% RSLogix 500 project Multiposition-Servo-Application.RSS, saved by version 8.30.00.16 %
PROJECT "UNTITLED"    % processor: Bul.1763 MicroLogix 1100 Series B %

PROGRAM FILES
  LAD 2 "MAIN"  4 rungs
  LAD 3 "IO"  7 rungs
  LAD 4 "CTRL"  10 rungs
  LAD 5 "POSI"  9 rungs

DATA FILES
  O0 OUTPUT  4 elements
  I1 INPUT  6 elements
  S2 STATUS  66 elements
  B3 BINARY  4 elements
  T4 TIMER  3 elements
  C5 COUNTER  1 elements
  R6 CONTROL  1 elements
  N7 INTEGER  2 elements
  F8 FLOAT  1 elements

LADDER 2 "MAIN"
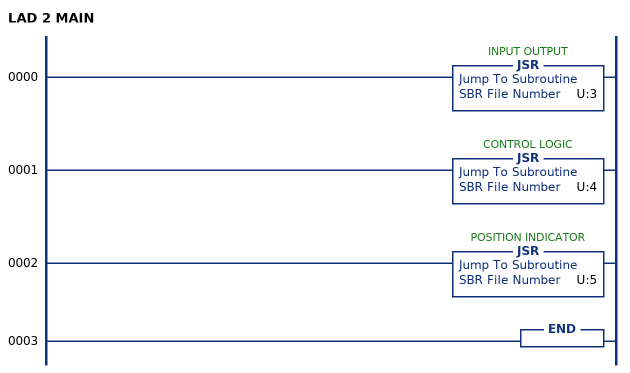
% Rung: 0 %
SOR JSR U:3 EOR
%   U:3  "INPUT OUTPUT" %
% Rung: 1 %
SOR JSR U:4 EOR
%   U:4  "CONTROL LOGIC" %
% Rung: 2 %
SOR JSR U:5 EOR
%   U:5  "POSITION INDICATOR" %
% Rung: 3 %
SOR END EOR

LADDER 3 "IO"
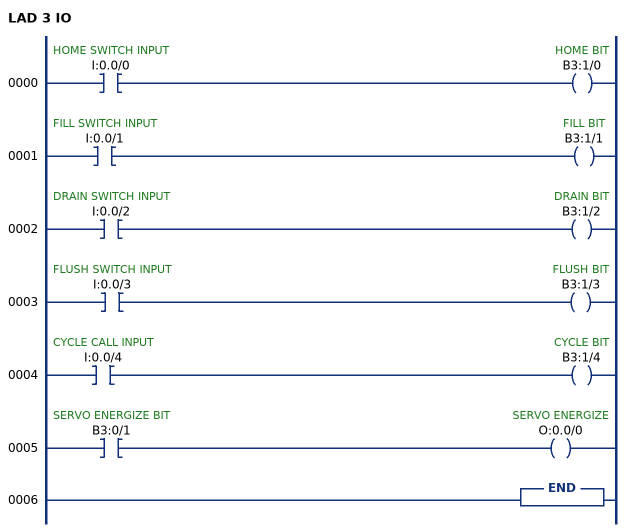
% Rung: 0 %
SOR XIC I:0.0/0 OTE B3:1/0 EOR
%   I:0.0/0  "HOME SWITCH INPUT" %
%   B3:1/0  "HOME BIT" %
% Rung: 1 %
SOR XIC I:0.0/1 OTE B3:1/1 EOR
%   I:0.0/1  "FILL SWITCH INPUT" %
%   B3:1/1  "FILL BIT" %
% Rung: 2 %
SOR XIC I:0.0/2 OTE B3:1/2 EOR
%   I:0.0/2  "DRAIN SWITCH INPUT" %
%   B3:1/2  "DRAIN BIT" %
% Rung: 3 %
SOR XIC I:0.0/3 OTE B3:1/3 EOR
%   I:0.0/3  "FLUSH SWITCH INPUT" %
%   B3:1/3  "FLUSH BIT" %
% Rung: 4 %
SOR XIC I:0.0/4 OTE B3:1/4 EOR
%   I:0.0/4  "CYCLE CALL INPUT" %
%   B3:1/4  "CYCLE BIT" %
% Rung: 5 %
SOR XIC B3:0/1 OTE O:0.0/0 EOR
%   B3:0/1  "SERVO ENERGIZE BIT" %
%   O:0.0/0  "SERVO ENERGIZE" %
% Rung: 6 %
SOR END EOR

LADDER 4 "CTRL"
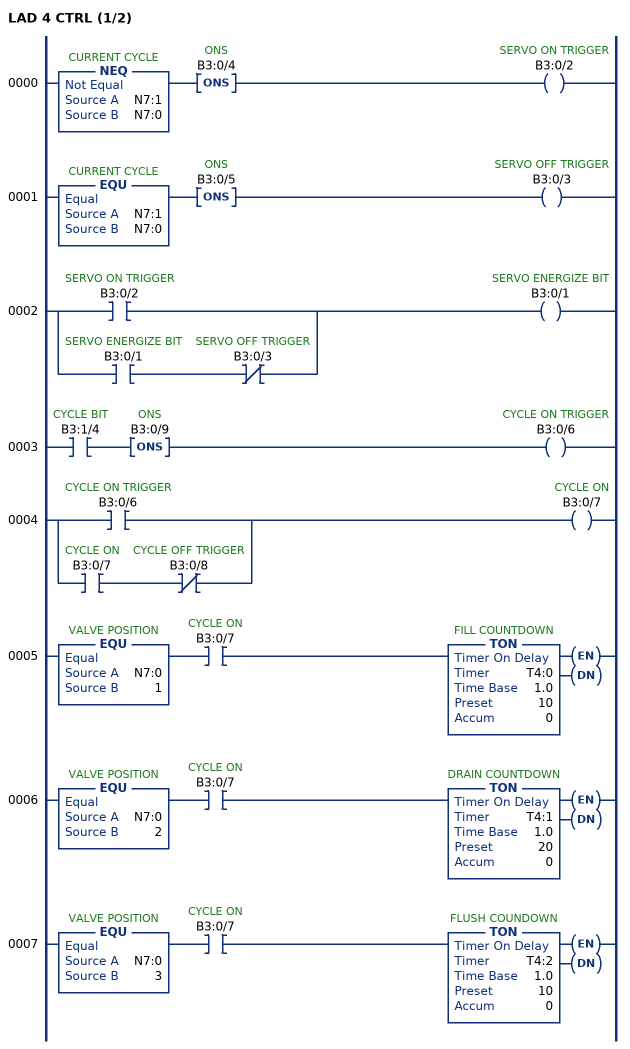
% Rung: 0 %
SOR NEQ N7:1 N7:0 ONS B3:0/4 OTE B3:0/2 EOR
%   N7:1  "CURRENT CYCLE" %
%   N7:0  "VALVE POSITION" %
%   B3:0/4  "ONS" %
%   B3:0/2  "SERVO ON TRIGGER" %
% Rung: 1 %
SOR EQU N7:1 N7:0 ONS B3:0/5 OTE B3:0/3 EOR
%   N7:1  "CURRENT CYCLE" %
%   N7:0  "VALVE POSITION" %
%   B3:0/5  "ONS" %
%   B3:0/3  "SERVO OFF TRIGGER" %
% Rung: 2 %
SOR BST XIC B3:0/2 NXB XIC B3:0/1 XIO B3:0/3 BND OTE B3:0/1 EOR
%   B3:0/2  "SERVO ON TRIGGER" %
%   B3:0/1  "SERVO ENERGIZE BIT" %
%   B3:0/3  "SERVO OFF TRIGGER" %
% Rung: 3 %
SOR XIC B3:1/4 ONS B3:0/9 OTE B3:0/6 EOR
%   B3:1/4  "CYCLE BIT" %
%   B3:0/9  "ONS" %
%   B3:0/6  "CYCLE ON TRIGGER" %
% Rung: 4 %
SOR BST XIC B3:0/6 NXB XIC B3:0/7 XIO B3:0/8 BND OTE B3:0/7 EOR
%   B3:0/6  "CYCLE ON TRIGGER" %
%   B3:0/7  "CYCLE ON" %
%   B3:0/8  "CYCLE OFF TRIGGER" %
% Rung: 5 %
SOR EQU N7:0 1 XIC B3:0/7 TON T4:0 1.0 10 0 EOR
%   N7:0  "VALVE POSITION" %
%   B3:0/7  "CYCLE ON" %
%   T4:0  "FILL COUNTDOWN" %
% Rung: 6 %
SOR EQU N7:0 2 XIC B3:0/7 TON T4:1 1.0 20 0 EOR
%   N7:0  "VALVE POSITION" %
%   B3:0/7  "CYCLE ON" %
%   T4:1  "DRAIN COUNTDOWN" %
% Rung: 7 %
SOR EQU N7:0 3 XIC B3:0/7 TON T4:2 1.0 10 0 EOR
%   N7:0  "VALVE POSITION" %
%   B3:0/7  "CYCLE ON" %
%   T4:2  "FLUSH COUNDOWN" %

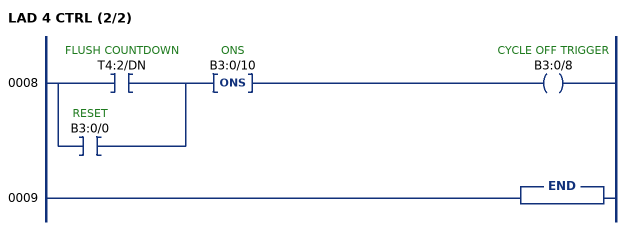
% Rung: 8 %
SOR BST XIC T4:2/DN NXB XIC B3:0/0 BND ONS B3:0/10 OTE B3:0/8 EOR
%   T4:2/DN  "FLUSH COUNTDOWN" %
%   B3:0/0  "RESET" %
%   B3:0/10  "ONS" %
%   B3:0/8  "CYCLE OFF TRIGGER" %
% Rung: 9 %
SOR END EOR

LADDER 5 "POSI"
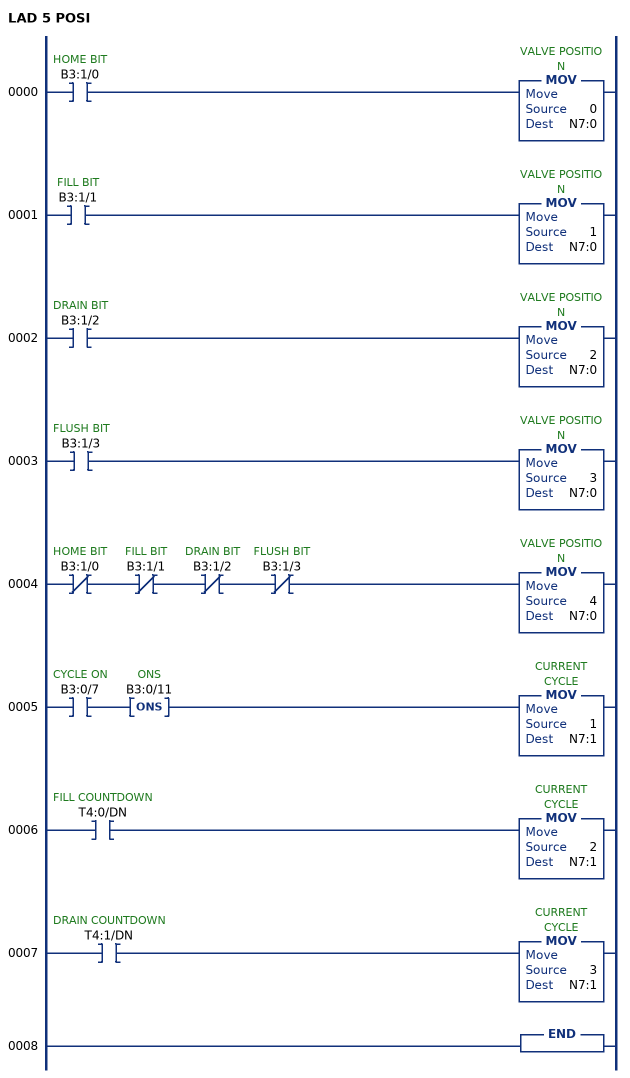
% Rung: 0 %
SOR XIC B3:1/0 MOV 0 N7:0 EOR
%   B3:1/0  "HOME BIT" %
%   N7:0  "VALVE POSITION" %
% Rung: 1 %
SOR XIC B3:1/1 MOV 1 N7:0 EOR
%   B3:1/1  "FILL BIT" %
%   N7:0  "VALVE POSITION" %
% Rung: 2 %
SOR XIC B3:1/2 MOV 2 N7:0 EOR
%   B3:1/2  "DRAIN BIT" %
%   N7:0  "VALVE POSITION" %
% Rung: 3 %
SOR XIC B3:1/3 MOV 3 N7:0 EOR
%   B3:1/3  "FLUSH BIT" %
%   N7:0  "VALVE POSITION" %
% Rung: 4 %
SOR XIO B3:1/0 XIO B3:1/1 XIO B3:1/2 XIO B3:1/3 MOV 4 N7:0 EOR
%   B3:1/0  "HOME BIT" %
%   B3:1/1  "FILL BIT" %
%   B3:1/2  "DRAIN BIT" %
%   B3:1/3  "FLUSH BIT" %
%   N7:0  "VALVE POSITION" %
% Rung: 5 %
SOR XIC B3:0/7 ONS B3:0/11 MOV 1 N7:1 EOR
%   B3:0/7  "CYCLE ON" %
%   B3:0/11  "ONS" %
%   N7:1  "CURRENT CYCLE" %
% Rung: 6 %
SOR XIC T4:0/DN MOV 2 N7:1 EOR
%   T4:0/DN  "FILL COUNTDOWN" %
%   N7:1  "CURRENT CYCLE" %
% Rung: 7 %
SOR XIC T4:1/DN MOV 3 N7:1 EOR
%   T4:1/DN  "DRAIN COUNTDOWN" %
%   N7:1  "CURRENT CYCLE" %
% Rung: 8 %
SOR END EOR

OTHER DOCUMENTED ADDRESSES
  B3:2/0  "ONS"
  B3:2/1  "ONS"
  B3:2/2  "ONS"
  B3:2/3  "CYCLE STARTED"
  B3:2/4  "ONS"
  B3:2/5  "ONS"

DATA TABLE (non-zero values as saved)
DATA T4
% .PRE .ACC %
% T4:0 % 10 0
% T4:1 % 20 0
% T4:2 % 10 0
